TYPE (* IEC61131-3, Table 14#5 *)
  (* Standard: 1131-3 *)
  (* Version 0.0, 1/8/2024, Cheyan, Schneider Electric, Template *)
  PACKAGE Main;
  {SET_ATTRIBUTE(nxtDataType, QdpEwqSPB7ofXswuXlSUf+xi5gGvP5fI9S3g9sPnd5F/ItQewYVETWVF32ZEpfDEbDXUqC6iYY3SUieZ6pgBGZ+JXQthypNoMwoEA3Z5oaKBFdqY+nG0rItTygy9uzM/EtK7RcrH5oXVGB9k67FawbPOH41NASKea4lJfaVuH7LwGY+SjfQuiYuEeGCHZUhWL6UhThn+ty3WZ96iso1N/hkjBrZsGIjw)}
  TimeQuality : STRUCT
    LeapSecondsKnown : BOOL;
    ClockFailure : BOOL;
    ClockNotSynchronized : BOOL;
    TimeAccuracy : TimeAccuracy;
  END_STRUCT;
END_TYPE
